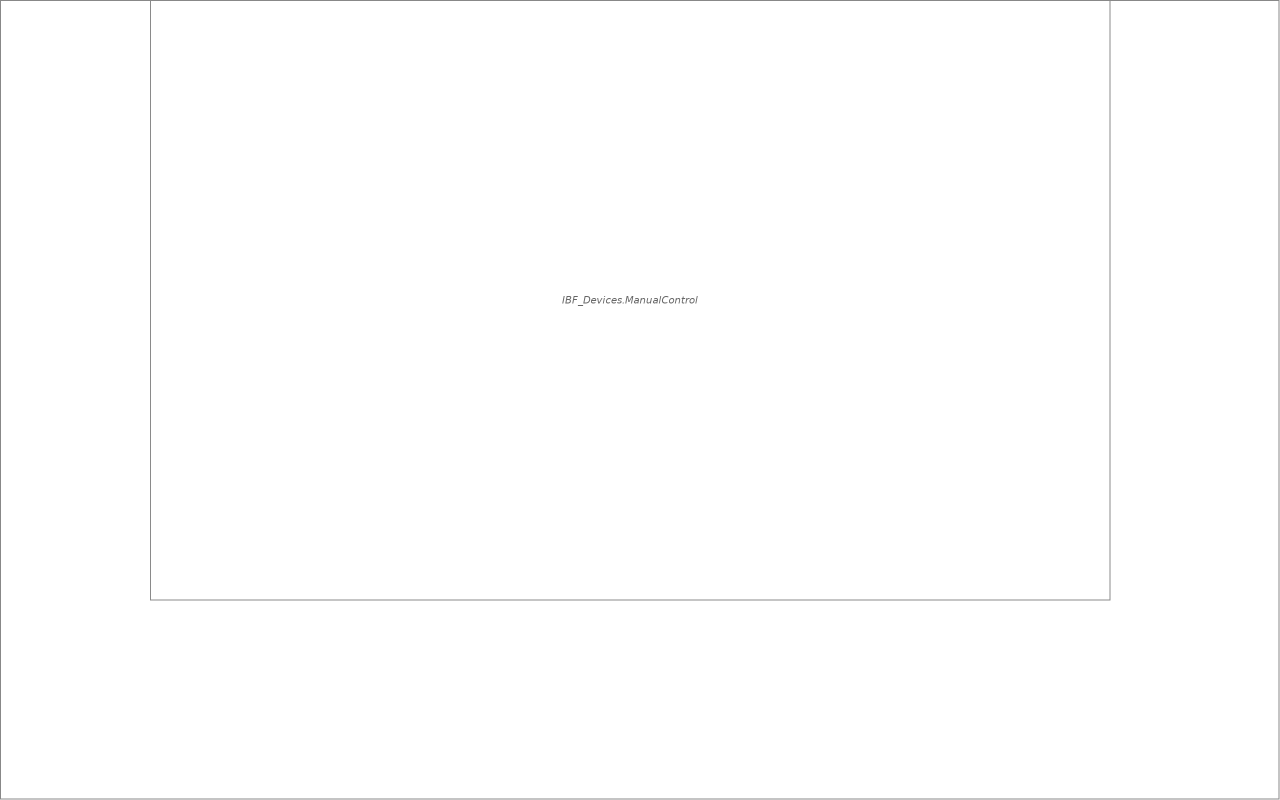
VISUALIZATION Manual  // 1280x800
    Frame (150,0 960x600)
        shows IBF_Devices.ManualControl(stHMI := GVL_DevManual.fbManualControler.stHMI, fbManualController := GVL_DevManual.fbManualControler)
END_VISUALIZATION

(* stored: Version 1.1.0.1, ProductVersion 3.1.4024.11
   Visu Manual: Id {8b12630b-f7fc-46df-9948-3293bcc3e0af} *)
